(* PLC project Sin nombre, Desconocido Sin nombre 1 *)
(* stored: creationDateTime 2025-06-16T20:32:46, modificationDateTime 2025-06-16T21:37:50 *)

PROGRAM Main
  VAR
    xFC_CERRADA AT %I0.0 : BOOL;
    xFC_BYPASS AT %I0.1 : BOOL;
    xFC_ABIERTA AT %I0.2 : BOOL;
    xApertura AT %I0.3 : BOOL;
    xPausa AT %I0.4 : BOOL;
    xCierre AT %I0.5 : BOOL;
    xQ_BOMBA AT %Q0.0 : BOOL;
    xQ_VALV_CIERRE AT %Q0.1 : BOOL;
    xPASO_3 AT %M0.2 : BOOL;
  END_VAR
  VAR
    Temp_Apertura : TON;
    Temp_Bloqueo : TON;
    Temp_Rearranque : TON;
  END_VAR

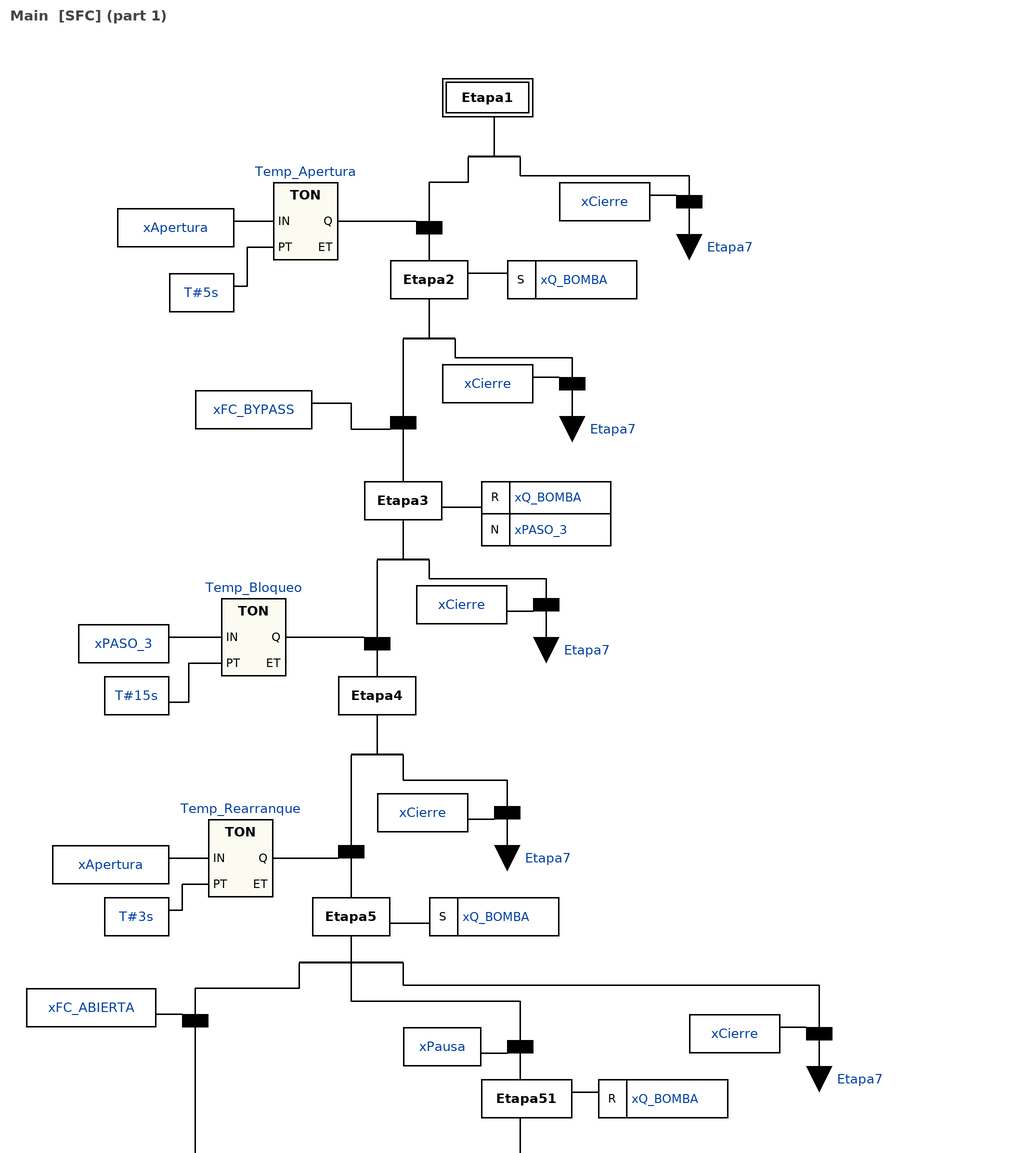
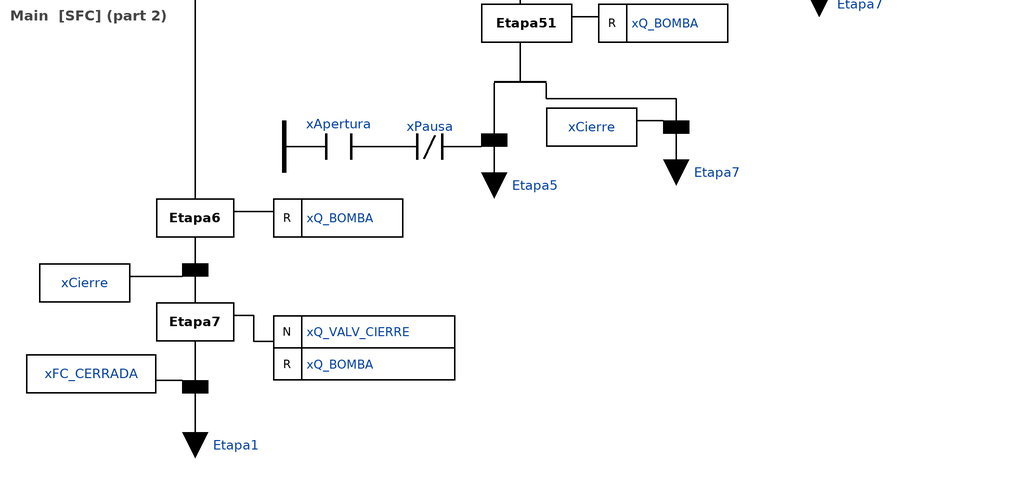
INITIAL_STEP Etapa1:
  COMPUTE_FUNCTION_BLOCKS(S);
END_STEP
TRANSITION FROM Etapa1 TO Etapa2
  := Temp_Apertura.Q;
END_TRANSITION
TRANSITION FROM Etapa1 TO Etapa7
  := xCierre;
END_TRANSITION
STEP Etapa2:
  xQ_BOMBA(S);
END_STEP
TRANSITION FROM Etapa2 TO Etapa3
  := xFC_BYPASS;
END_TRANSITION
TRANSITION FROM Etapa2 TO Etapa7
  := xCierre;
END_TRANSITION
STEP Etapa3:
  xQ_BOMBA(R);
  xPASO_3(N);
END_STEP
TRANSITION FROM Etapa3 TO Etapa4
  := Temp_Bloqueo.Q;
END_TRANSITION
TRANSITION FROM Etapa3 TO Etapa7
  := xCierre;
END_TRANSITION
STEP Etapa4:
END_STEP
TRANSITION FROM Etapa4 TO Etapa5
  := Temp_Rearranque.Q;
END_TRANSITION
TRANSITION FROM Etapa4 TO Etapa7
  := xCierre;
END_TRANSITION
STEP Etapa5:
  xQ_BOMBA(S);
END_STEP
TRANSITION FROM Etapa5 TO Etapa51
  := xPausa;
END_TRANSITION
TRANSITION FROM Etapa5 TO Etapa6
  := xFC_ABIERTA;
END_TRANSITION
TRANSITION FROM Etapa5 TO Etapa7
  := xCierre;
END_TRANSITION
STEP Etapa51:
  xQ_BOMBA(R);
END_STEP
TRANSITION FROM Etapa51 TO Etapa5
  := xApertura AND NOT xPausa;
END_TRANSITION
TRANSITION FROM Etapa51 TO Etapa7
  := xCierre;
END_TRANSITION
STEP Etapa6:
  xQ_BOMBA(R);
END_STEP
TRANSITION FROM Etapa6 TO Etapa7
  := xCierre;
END_TRANSITION
STEP Etapa7:
  xQ_VALV_CIERRE(N);
  xQ_BOMBA(R);
END_STEP
TRANSITION FROM Etapa7 TO Etapa1
  := xFC_CERRADA;
END_TRANSITION
ACTION COMPUTE_FUNCTION_BLOCKS:  (* blocks drawn on the SFC sheet *)
  Temp_Apertura(IN := xApertura, PT := T#5s);
  Temp_Bloqueo(IN := xPASO_3, PT := T#15s);
  Temp_Rearranque(IN := xApertura, PT := T#3s);
END_ACTION
END_PROGRAM

CONFIGURATION Config0
  RESOURCE Res0 ON PLC
    TASK task0(INTERVAL := T#20ms, PRIORITY := 0);
    PROGRAM instance0 WITH task0 : Main;
  END_RESOURCE
END_CONFIGURATION
